{attribute 'GeneratedUsingTerminal: EK1100-0000-0018'}
{attribute addProperty BoxType "EK1100-0000-0018"}
{attribute addProperty Id "Beckhoff_EL6xxxEK1122Beckhoff_EL6xxxEK1122_B6505ABE2A_0001_EL6001_0000_0000EL6001_C5ADEF9E60A_0002_EL6001_0000_0016EL6001_B592E1CA69A_0003_EL6001_0000_0017EL6001_B592E1CA69A_0004_EL6001_0000_0018EL6001_B592E1CA69A_0005_EL6001_0000_0019EL6001_B592E1CA69A_0006_EL6001_0000_0020EL6001_B592E1CA69A_0007_EL6002_0000_0016EL6002_D5B468BD126A_0008_EL6002_0000_0017EL6002_81703A53126A_0009_EL6002_0000_0018EL6002_81703A53126A_0010_EL6002_0000_0019EL6002_81703A53126A_0011_EL6021_0000_0000EL6021_C5ADEF9E60A_0012_EL6021_0000_0016EL6021_B592E1CA69A_0013_EL6021_0000_0017EL6021_B592E1CA69A_0014_EL6021_0000_0018EL6021_4CB9967B69A_0015_EL6021_0000_0019EL6021_4CB9967B69A_0016_EL6021_0000_0020EL6021_4CB9967B69A_0017_EL6021_0000_0021EL6021_4CB9967B69A_0018_EL6021_0021_0018EL6021_4CB9967B69A_0019_EL6021_0021_0019EL6021_4CB9967B69A_0020_EL6021_0021_0020EL6021_4CB9967B69A_0021_EL6021_0021_0021EL6021_4CB9967B69A_0022_EL6022_0000_0016EL6022_D5B468BD126A_0023_EL6022_0000_0017EL6022_D5B468BD126A_0024_EL6022_0000_0018EL6022_D5B468BD126A_0025_EL6022_0000_0019EL6022_D5B468BD126A_0026_EL6070_0000_0016EL6070_EEB2FEF410A_0027_EL6070_0000_0017EL6070_EEB2FEF410A_0028_EL6070_0000_0018EL6070_EEB2FEF410A_0029_EL6070_0000_0019EL6070_EEB2FEF410A_0030_EL6070_0033_0016EL6070_EEB2FEF410A_0031_EL6070_0033_0017EL6070_EEB2FEF410A_0032_EL6070_0033_0018EL6070_EEB2FEF410A_0033_EL6070_0033_0019EL6070_EEB2FEF410A_0034_EL6080_0000_0016EL6080_BB2AF53012A_0035_EL6080_0000_0017EL6080_BB2AF53012A_0036_EL6080_0000_0018EL6080_9D61BA3F16A_0037_EL6080_0000_0020EL6080_9D61BA3F16A_0038_EL6090_0000_0016EL6090_18BD01E922A_0039_EL6090_0000_0017EL6090_18BD01E922A_0040_EL6201_0000_0017EL6201_12FC4F5D524A_0041_EL6201_0000_0018EL6201_F71597F7528A_0042_EL6201_0000_0019EL6201_F71597F7528A_0043_EL6224_0000_0016EL6224_DFFBB70222A_0044_EL6224_0000_0017EL6224_EDFF9F2F24A_0045_EL6224_0000_0018EL6224_EDFF9F2F24A_0046_EL6224_0000_0019EL6224_EDFF9F2F24A_0047_EL6224_0000_0020EL6224_EDFF9F2F24A_0048_EL6224_0000_0021EL6224_EDFF9F2F24A_0049_EL6224_0090_0016EL6224_98EF241924A_0050_EL6224_0090_0017EL6224_98EF241924"}
{attribute addProperty CRC "1479734440"}
{attribute addProperty Size "4115"}
TYPE Beckhoff_EL6xxx_5832F4A8 EXTENDS EK1100_1FC0878B :
STRUCT
	{attribute addProperty Name "Beckhoff EL6xxxEK1122"}
	{attribute addProperty PreviousPort "Beckhoff EL6xxx : B"}
	Beckhoff_EL6xxxEK1122 : Beckhoff_EL6xxxEK1122_B6505ABE;
	{attribute addProperty Name "A_0001(EL6001-0000-0000)"}
	{attribute addProperty PreviousPort "Beckhoff EL6xxxEK1122 : C"}
	A_0001_EL6001_0000_0000 : EL6001_C5ADEF9E;
	{attribute addProperty Name "A_0002(EL6001-0000-0016)"}
	{attribute addProperty PreviousPort "A_0001(EL6001-0000-0000) : B"}
	A_0002_EL6001_0000_0016 : EL6001_B592E1CA;
	{attribute addProperty Name "A_0003(EL6001-0000-0017)"}
	{attribute addProperty PreviousPort "A_0002(EL6001-0000-0016) : B"}
	A_0003_EL6001_0000_0017 : EL6001_B592E1CA;
	{attribute addProperty Name "A_0004(EL6001-0000-0018)"}
	{attribute addProperty PreviousPort "A_0003(EL6001-0000-0017) : B"}
	A_0004_EL6001_0000_0018 : EL6001_B592E1CA;
	{attribute addProperty Name "A_0005(EL6001-0000-0019)"}
	{attribute addProperty PreviousPort "A_0004(EL6001-0000-0018) : B"}
	A_0005_EL6001_0000_0019 : EL6001_B592E1CA;
	{attribute addProperty Name "A_0006(EL6001-0000-0020)"}
	{attribute addProperty PreviousPort "A_0005(EL6001-0000-0019) : B"}
	A_0006_EL6001_0000_0020 : EL6001_B592E1CA;
	{attribute addProperty Name "A_0007(EL6002-0000-0016)"}
	{attribute addProperty PreviousPort "A_0006(EL6001-0000-0020) : B"}
	A_0007_EL6002_0000_0016 : EL6002_D5B468BD;
	{attribute addProperty Name "A_0008(EL6002-0000-0017)"}
	{attribute addProperty PreviousPort "A_0007(EL6002-0000-0016) : B"}
	A_0008_EL6002_0000_0017 : EL6002_81703A53;
	{attribute addProperty Name "A_0009(EL6002-0000-0018)"}
	{attribute addProperty PreviousPort "A_0008(EL6002-0000-0017) : B"}
	A_0009_EL6002_0000_0018 : EL6002_81703A53;
	{attribute addProperty Name "A_0010(EL6002-0000-0019)"}
	{attribute addProperty PreviousPort "A_0009(EL6002-0000-0018) : B"}
	A_0010_EL6002_0000_0019 : EL6002_81703A53;
	{attribute addProperty Name "A_0011(EL6021-0000-0000)"}
	{attribute addProperty PreviousPort "A_0010(EL6002-0000-0019) : B"}
	A_0011_EL6021_0000_0000 : EL6021_C5ADEF9E;
	{attribute addProperty Name "A_0012(EL6021-0000-0016)"}
	{attribute addProperty PreviousPort "A_0011(EL6021-0000-0000) : B"}
	A_0012_EL6021_0000_0016 : EL6021_B592E1CA;
	{attribute addProperty Name "A_0013(EL6021-0000-0017)"}
	{attribute addProperty PreviousPort "A_0012(EL6021-0000-0016) : B"}
	A_0013_EL6021_0000_0017 : EL6021_B592E1CA;
	{attribute addProperty Name "A_0014(EL6021-0000-0018)"}
	{attribute addProperty PreviousPort "A_0013(EL6021-0000-0017) : B"}
	A_0014_EL6021_0000_0018 : EL6021_4CB9967B;
	{attribute addProperty Name "A_0015(EL6021-0000-0019)"}
	{attribute addProperty PreviousPort "A_0014(EL6021-0000-0018) : B"}
	A_0015_EL6021_0000_0019 : EL6021_4CB9967B;
	{attribute addProperty Name "A_0016(EL6021-0000-0020)"}
	{attribute addProperty PreviousPort "A_0015(EL6021-0000-0019) : B"}
	A_0016_EL6021_0000_0020 : EL6021_4CB9967B;
	{attribute addProperty Name "A_0017(EL6021-0000-0021)"}
	{attribute addProperty PreviousPort "A_0016(EL6021-0000-0020) : B"}
	A_0017_EL6021_0000_0021 : EL6021_4CB9967B;
	{attribute addProperty Name "A_0018(EL6021-0021-0018)"}
	{attribute addProperty PreviousPort "A_0017(EL6021-0000-0021) : B"}
	A_0018_EL6021_0021_0018 : EL6021_4CB9967B;
	{attribute addProperty Name "A_0019(EL6021-0021-0019)"}
	{attribute addProperty PreviousPort "A_0018(EL6021-0021-0018) : B"}
	A_0019_EL6021_0021_0019 : EL6021_4CB9967B;
	{attribute addProperty Name "A_0020(EL6021-0021-0020)"}
	{attribute addProperty PreviousPort "A_0019(EL6021-0021-0019) : B"}
	A_0020_EL6021_0021_0020 : EL6021_4CB9967B;
	{attribute addProperty Name "A_0021(EL6021-0021-0021)"}
	{attribute addProperty PreviousPort "A_0020(EL6021-0021-0020) : B"}
	A_0021_EL6021_0021_0021 : EL6021_4CB9967B;
	{attribute addProperty Name "A_0022(EL6022-0000-0016)"}
	{attribute addProperty PreviousPort "A_0021(EL6021-0021-0021) : B"}
	A_0022_EL6022_0000_0016 : EL6022_D5B468BD;
	{attribute addProperty Name "A_0023(EL6022-0000-0017)"}
	{attribute addProperty PreviousPort "A_0022(EL6022-0000-0016) : B"}
	A_0023_EL6022_0000_0017 : EL6022_D5B468BD;
	{attribute addProperty Name "A_0024(EL6022-0000-0018)"}
	{attribute addProperty PreviousPort "A_0023(EL6022-0000-0017) : B"}
	A_0024_EL6022_0000_0018 : EL6022_D5B468BD;
	{attribute addProperty Name "A_0025(EL6022-0000-0019)"}
	{attribute addProperty PreviousPort "A_0024(EL6022-0000-0018) : B"}
	A_0025_EL6022_0000_0019 : EL6022_D5B468BD;
	{attribute addProperty Name "A_0026(EL6070-0000-0016)"}
	{attribute addProperty PreviousPort "A_0025(EL6022-0000-0019) : B"}
	A_0026_EL6070_0000_0016 : EL6070_EEB2FEF4;
	{attribute addProperty Name "A_0027(EL6070-0000-0017)"}
	{attribute addProperty PreviousPort "A_0026(EL6070-0000-0016) : B"}
	A_0027_EL6070_0000_0017 : EL6070_EEB2FEF4;
	{attribute addProperty Name "A_0028(EL6070-0000-0018)"}
	{attribute addProperty PreviousPort "A_0027(EL6070-0000-0017) : B"}
	A_0028_EL6070_0000_0018 : EL6070_EEB2FEF4;
	{attribute addProperty Name "A_0029(EL6070-0000-0019)"}
	{attribute addProperty PreviousPort "A_0028(EL6070-0000-0018) : B"}
	A_0029_EL6070_0000_0019 : EL6070_EEB2FEF4;
	{attribute addProperty Name "A_0030(EL6070-0033-0016)"}
	{attribute addProperty PreviousPort "A_0029(EL6070-0000-0019) : B"}
	A_0030_EL6070_0033_0016 : EL6070_EEB2FEF4;
	{attribute addProperty Name "A_0031(EL6070-0033-0017)"}
	{attribute addProperty PreviousPort "A_0030(EL6070-0033-0016) : B"}
	A_0031_EL6070_0033_0017 : EL6070_EEB2FEF4;
	{attribute addProperty Name "A_0032(EL6070-0033-0018)"}
	{attribute addProperty PreviousPort "A_0031(EL6070-0033-0017) : B"}
	A_0032_EL6070_0033_0018 : EL6070_EEB2FEF4;
	{attribute addProperty Name "A_0033(EL6070-0033-0019)"}
	{attribute addProperty PreviousPort "A_0032(EL6070-0033-0018) : B"}
	A_0033_EL6070_0033_0019 : EL6070_EEB2FEF4;
	{attribute addProperty Name "A_0034(EL6080-0000-0016)"}
	{attribute addProperty PreviousPort "A_0033(EL6070-0033-0019) : B"}
	A_0034_EL6080_0000_0016 : EL6080_BB2AF530;
	{attribute addProperty Name "A_0035(EL6080-0000-0017)"}
	{attribute addProperty PreviousPort "A_0034(EL6080-0000-0016) : B"}
	A_0035_EL6080_0000_0017 : EL6080_BB2AF530;
	{attribute addProperty Name "A_0036(EL6080-0000-0018)"}
	{attribute addProperty PreviousPort "A_0035(EL6080-0000-0017) : B"}
	A_0036_EL6080_0000_0018 : EL6080_9D61BA3F;
	{attribute addProperty Name "A_0037(EL6080-0000-0020)"}
	{attribute addProperty PreviousPort "A_0036(EL6080-0000-0018) : B"}
	A_0037_EL6080_0000_0020 : EL6080_9D61BA3F;
	{attribute addProperty Name "A_0038(EL6090-0000-0016)"}
	{attribute addProperty PreviousPort "A_0037(EL6080-0000-0020) : B"}
	A_0038_EL6090_0000_0016 : EL6090_18BD01E9;
	{attribute addProperty Name "A_0039(EL6090-0000-0017)"}
	{attribute addProperty PreviousPort "A_0038(EL6090-0000-0016) : B"}
	A_0039_EL6090_0000_0017 : EL6090_18BD01E9;
	{attribute addProperty Name "A_0040(EL6201-0000-0017)"}
	{attribute addProperty PreviousPort "A_0039(EL6090-0000-0017) : B"}
	A_0040_EL6201_0000_0017 : EL6201_12FC4F5D;
	{attribute addProperty Name "A_0041(EL6201-0000-0018)"}
	{attribute addProperty PreviousPort "A_0040(EL6201-0000-0017) : B"}
	A_0041_EL6201_0000_0018 : EL6201_F71597F7;
	{attribute addProperty Name "A_0042(EL6201-0000-0019)"}
	{attribute addProperty PreviousPort "A_0041(EL6201-0000-0018) : B"}
	A_0042_EL6201_0000_0019 : EL6201_F71597F7;
	{attribute addProperty Name "A_0043(EL6224-0000-0016)"}
	{attribute addProperty PreviousPort "A_0042(EL6201-0000-0019) : B"}
	A_0043_EL6224_0000_0016 : EL6224_DFFBB702;
	{attribute addProperty Name "A_0044(EL6224-0000-0017)"}
	{attribute addProperty PreviousPort "A_0043(EL6224-0000-0016) : B"}
	A_0044_EL6224_0000_0017 : EL6224_EDFF9F2F;
	{attribute addProperty Name "A_0045(EL6224-0000-0018)"}
	{attribute addProperty PreviousPort "A_0044(EL6224-0000-0017) : B"}
	A_0045_EL6224_0000_0018 : EL6224_EDFF9F2F;
	{attribute addProperty Name "A_0046(EL6224-0000-0019)"}
	{attribute addProperty PreviousPort "A_0045(EL6224-0000-0018) : B"}
	A_0046_EL6224_0000_0019 : EL6224_EDFF9F2F;
	{attribute addProperty Name "A_0047(EL6224-0000-0020)"}
	{attribute addProperty PreviousPort "A_0046(EL6224-0000-0019) : B"}
	A_0047_EL6224_0000_0020 : EL6224_EDFF9F2F;
	{attribute addProperty Name "A_0048(EL6224-0000-0021)"}
	{attribute addProperty PreviousPort "A_0047(EL6224-0000-0020) : B"}
	A_0048_EL6224_0000_0021 : EL6224_EDFF9F2F;
	{attribute addProperty Name "A_0049(EL6224-0090-0016)"}
	{attribute addProperty PreviousPort "A_0048(EL6224-0000-0021) : B"}
	A_0049_EL6224_0090_0016 : EL6224_98EF2419;
	{attribute addProperty Name "A_0050(EL6224-0090-0017)"}
	{attribute addProperty PreviousPort "A_0049(EL6224-0090-0016) : B"}
	A_0050_EL6224_0090_0017 : EL6224_98EF2419;
END_STRUCT
END_TYPE

(* stored: Version 1.2.0.0, ProductVersion 3.1.4024.11
   DUT Beckhoff_EL6xxx_5832F4A8: Id {cb7d69e1-4650-4f2b-91ef-6eddd21d4008} *)
